TYPE ST_PowerDemand :
STRUCT
	b_Demand_24V	:	BOOL;
	b_Demand_400V	:	BOOL;
	b_Demand_HVDC	:	BOOL;
END_STRUCT
END_TYPE

(* stored: Version 1.1.0.1, ProductVersion 3.1.4024.12
   DUT ST_PowerDemand: Id {434479ad-f678-4d4c-926d-ec343f545ffd} *)
